TYPE motor_state_datagrid :
STRUCT
	state : INT;
END_STRUCT
END_TYPE

(* stored: Version 1.1.0.1, ProductVersion 3.1.4024.12
   DUT motor_state_datagrid: Id {133a0835-1cbd-433c-b8b5-b94605bcfdd4} *)
